(* PLC project ArduinoNano, Desconhecido Sem nome 1 *)
(* stored: creationDateTime 2025-10-30T20:05:32, modificationDateTime 2025-10-30T21:34:14 *)

PROGRAM potenciometro
  VAR
    pot_valor AT %IW1 : UINT;  (* pino A1 *)
  END_VAR
  VAR
    ref : UINT := 32767;  (* referência *)
  END_VAR
  VAR
    led_saida AT %QX0.3 : BOOL;  (* pino D13 *)
  END_VAR

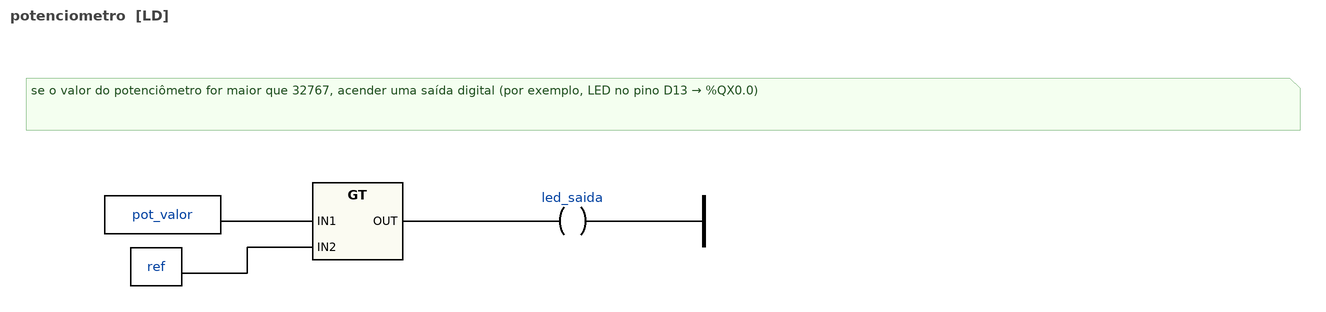
(* LD diagram, written out as Structured Text *)
(* se o valor do potenciômetro for maior que 32767, acender uma saída digital (por exemplo, LED no pino D13 → %QX0.0) *)
led_saida := pot_valor > ref;
END_PROGRAM

CONFIGURATION Config0
  RESOURCE Res0 ON PLC
    TASK task0(INTERVAL := T#20ms, PRIORITY := 0);
    PROGRAM instance0 WITH task0 : potenciometro;
  END_RESOURCE
END_CONFIGURATION
